Staubli VAL3: CartesianSpace.pjx

--- CartesianSpace.pjx ---
Parameters version=s7.9.1 stackSize=5000 millimeterUnit=true
Data file=CartesianSpace.dtx
Type name=CartesianPos path=./CartesianPos/CartesianPos.pjx
Type name=CartesianVel path=./CartesianVel/CartesianVel.pjx
Type name=CartesianAccel path=./CartesianAccel/CartesianAccel.pjx
Type name=CartesianForce path=./CartesianForce/CartesianForce.pjx

--- CartesianSpace.dtx ---
public CartesianPos cartesianPos
  [0]
    pointRx cp
public CartesianVel cartesianVel
  [0]
    num resVel
    num cv[6]
public CartesianAccel cartesianAccel
  [0]
    num ca[6]
    num resAccel
public CartesianForce cartesianForce
  [0]
    num cf[6]
    num resForce
